FUNCTION_BLOCK ARRAY2VALUES_2_LREAL
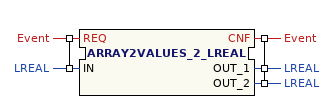
  EVENT_INPUT
    REQ WITH IN;
  END_EVENT
  EVENT_OUTPUT
    CNF WITH OUT_1, OUT_2;
  END_EVENT
  VAR_INPUT
    IN : LREAL;
  END_VAR
  VAR_OUTPUT
    OUT_1 : LREAL;
    OUT_2 : LREAL;
  END_VAR
END_FUNCTION_BLOCK
